{attribute 'linkalways'} 
{attribute 'no_explicit_call' := 'This FB is a CLASS and must be accessed using methods or properties'}
{attribute 'enable_dynamic_creation'}
FUNCTION_BLOCK FINAL Node_FIND EXTENDS Node
VAR
	str1 : _STRING('');
	str2 : _STRING('');
	out : _INT(0);
END_VAR

METHOD PUBLIC  Clone : I_Node
VAR
	pNode : POINTER TO Node_FIND;
END_VAR
pNode := __NEW(Node_FIND);
Clone := pNode^;
END_METHOD

METHOD FB_init : BOOL
VAR_INPUT
	bInitRetains : BOOL; // if TRUE, the retain variables are initialized (warm start / cold start)
	bInCopyCode : BOOL;  // if TRUE, the instance afterwards gets moved into the copy code (online change)
END_VAR
AddParameter('str1', str1);
AddParameter('str2', str2);
AddOutput('out', out);
END_METHOD

METHOD PROTECTED OnExecute
VAR
END_VAR
out.Value := FIND(str1.Value, str2.Value);
END_METHOD

END_FUNCTION_BLOCK

(* stored: Version 1.1.0.1, ProductVersion 3.1.4026.18
   POU Node_FIND: Id {9c415066-01c4-023c-1458-77be78cbee75}, SpecialFunc None
   Folder Constructor: Id {24069f88-28ab-0942-044c-d1e0aed929d7}
   Method Clone: Id {574719c5-043f-0e6a-159b-856a104e74e1}
   Method FB_init: Id {5780ae02-39a5-00b4-0c55-7ff3a49e1370}
   Method OnExecute: Id {23bc0590-eb31-0c7c-269c-057fc1f4b68d} *)
